// TIA Portal V20 export
DATA_BLOCK "Simulation_DB"   // DB40118
// stored: InstanceOfName Unit1.Em11.Simulation, InstanceOfType FB, Namespace Unit1.Em11
"Unit1.Em11.Simulation"
   // VAR_INPUT
   //    simulation { ExternalAccessible := 'False'; ExternalVisible := 'False'; ExternalWritable := 'False'} : Bool;
   // END_VAR
   // VAR
   //    statDigitalSignal { ExternalAccessible := 'False'; ExternalVisible := 'False'; ExternalWritable := 'False'} : Array[0..9] of Bool;
   // END_VAR
BEGIN
END_DATA_BLOCK
